// LS Electric XG5000 project: test
// PLC NewPLC

PROGRAM NewProgram (task: 스캔 프로그램)

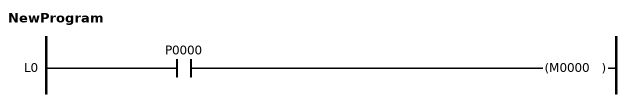
; L0
LOAD      P0000
OUT       M0000